FUNCTION_BLOCK T_TcpClientConnection
VAR
    connection : FB_ClientServerConnection;
	_log : T_NamedBase;
END_VAR

METHOD PUBLIC Connect
VAR_INPUT
  ip : T_IPv4Addr;
  port : UINT;
  timeout : TIME;
END_VAR
connection.sRemoteHost := ip;
connection.nRemotePort := port;
connection.tReconnect := timeout;
connection.nMode := CONNECT_MODE_ENABLEDBG;
connection.bEnable := TRUE;
END_METHOD

METHOD PUBLIC CyclicLogic
VAR_INST
	TON_ConnectTimer : TON;
END_VAR
connection();

TON_ConnectTimer(
	IN:= connection.bEnable AND NOT IsConnected,
	PT:= connection.tReconnect,
	Q=> ,
	ET=> );

IF TON_ConnectTimer.Q THEN
	connection.bEnable := FALSE;
	_log.LogError('Connection time out');
END_IF
END_METHOD

METHOD PUBLIC Disconnect
connection.bEnable := FALSE;
_log.LogInfo('Disconnected');
END_METHOD

PROPERTY ErrID : UDINT
GET
ErrID := connection.nErrId;
END_GET
END_PROPERTY

PROPERTY PUBLIC IsBusy : BOOL
GET
IsBusy := connection.bBusy;
END_GET
END_PROPERTY

PROPERTY PUBLIC IsConnected : BOOL
GET
IsConnected := (connection.eState = E_SocketConnectionState.eSOCKET_CONNECTED);
END_GET
END_PROPERTY

PROPERTY PUBLIC IsError : BOOL
GET
IsError := connection.bError;
END_GET
END_PROPERTY

PROPERTY PUBLIC Socket : REFERENCE TO T_HSOCKET
GET
Socket REF= connection.hSocket;
END_GET
END_PROPERTY

END_FUNCTION_BLOCK

(* stored: Version 1.1.0.1
   POU T_TcpClientConnection: Id {eaea54c5-977f-4611-9c99-b17f35128b8f}, SpecialFunc None
   Folder Methods: Id {6def861a-62b9-4c4c-8f17-7029d4004938}
   Folder Properties: Id {b0340ce8-3eeb-41a7-8440-33a147d8ba6f}
   Method Connect: Id {31913ce7-d64c-4dd7-9523-4cb6ecca04b5}
   Method CyclicLogic: Id {02f5bf77-288e-4841-bc8a-aeb4ef2ec743}
   Method Disconnect: Id {bcd1c9b6-20ca-4c90-a7ba-6571ffceca61}
   Property ErrID: Id {4c01374e-e118-4533-8afe-8def69b515e2}
   Get Get: Id {f633004f-cd87-4d79-82f3-96c15c67de5a}
   Property IsBusy: Id {2ffc28c2-c438-431b-8332-675d6f38478f}
   Get Get: Id {440d0775-bbcd-4244-9291-a0fc6df5ed93}
   Property IsConnected: Id {12af8a5f-3124-4214-b0f5-fb87bd44f1df}
   Get Get: Id {ab05c78f-5be3-4326-b844-b58c9d079910}
   Property IsError: Id {4facca61-76db-435c-a031-78ba8e61588a}
   Get Get: Id {a55f6aee-c8ea-4860-93df-67409f9f55d7}
   Property Socket: Id {700ebf11-fa88-4edf-97de-f19d67168f0f}
   Get Get: Id {7b1a6841-b485-47e9-960c-95973eb75e36} *)
